// TIA Portal V20 export
FUNCTION_BLOCK "FB_Gripper"   // FB54, SCL
{ S7_Optimized_Access := 'TRUE' }
// stored: MemoryReserve 100, SetENOAutomatically false
   VAR_INPUT
      iHoldPart : Bool;   // Hold Part Request
      iOpen : Bool;   // Shim Plate Opened (DI)
      iCloseWithoutPart : Bool;   // Shim Plate Closed with Part (DI)
      iPulseTime : Time;   // Pulse before Closing Time (WFA ???)
      iMonitorTime : Time;
   END_VAR
   VAR_OUTPUT
      oClose : Bool;   // Closing Request (DO)
      oOpen : Bool;   // Openeing Request (DO)
      oStateOpen : Bool;   // Opened Status
      oStateClose : Bool;   // Closed Status
      oStateCloseWithPart : Bool;   // Closed with Part Status
      oErrorCode { ExternalAccessible := 'False'; ExternalVisible := 'False'; ExternalWritable := 'False'} : Int;
   END_VAR
   VAR
      sPulseTimer : TP_TIME;   // Pulse before Closing Timer (WFA ???)
      sMonitorTimer : TON_TIME;
   END_VAR
BEGIN
   REGION Description header 
       //==================================================================================
       // POSALUX Swiss SA / (C) Copyright 2025
       //----------------------------------------------------------------------------------
       // Title: Initialization of axis
       // Comment/Function: FB_LoaderShimPlate
       // Author: Fabien WALDT
       // Engineering: TIA Portal v17
       //----------------------------------------------------------------------------------
       // Change log table:
       // Version  | Date     | Expert in charge | Changes applied
       // ---------|----------|------------------|-----------------------------------------
       // 00.00.01 | 20250423 | WFA              | First released version
       // =================================================================================
   END_REGION

   REGION Open - Close request
       // Close request
       #sPulseTimer(IN := #iHoldPart,
                   PT := #iPulseTime);
       #oClose := #sPulseTimer.Q AND #iHoldPart;

       // Open Request
       #oOpen := NOT #iHoldPart AND NOT #iOpen;
   END_REGION

   REGION Gripper States
       // State : Open
       #oStateOpen := #iOpen;

       //State : Close
       #oStateClose := NOT #iOpen AND NOT #oOpen AND NOT #oClose AND #iCloseWithoutPart ;

       // State : Close with Part
       #oStateCloseWithPart := NOT #iOpen AND NOT #oOpen AND NOT #oClose AND NOT #iCloseWithoutPart;
   END_REGION

   REGION Monitoring Timer
       #sMonitorTimer(IN := (#oOpen AND NOT #oStateOpen) OR
                      (#oClose AND (NOT #oStateClose AND NOT #oStateCloseWithPart) OR
                      (NOT #oStateOpen AND NOT #oStateClose AND NOT #oStateCloseWithPart) OR
                      (#oStateOpen AND (#oStateClose OR #oStateCloseWithPart))),
                      PT := #iMonitorTime);
   END_REGION

   REGION Error Codes
       #oErrorCode := 0;        // Code 0: No Error
       IF #oOpen AND #sMonitorTimer.Q THEN
           #oErrorCode := 1;    // Code 1: Error Open Command Plus
       ELSIF #oClose AND #sMonitorTimer.Q THEN
           #oErrorCode := 2;    // Code 2: Error Close Command Minus
       ELSIF NOT #oStateOpen AND NOT #oStateClose AND NOT #oStateCloseWithPart AND #sMonitorTimer.Q THEN
           #oErrorCode := 3;    // Code 3: Error Timeout Position OFF   
       ELSIF #oStateOpen AND (#oStateClose OR #oStateCloseWithPart) AND #sMonitorTimer.Q THEN
           #oErrorCode := 4;    // Code 4: Error Timeout Position ON       
       END_IF;
   END_REGION
END_FUNCTION_BLOCK
